// TwinCAT 3 PLC project Main
// ProgramVersion: 3.1.4024.0
// libraries:
//   mobject-core, * (mobject)
//   mobject-graph, * (mobject)
//   mobject-graph-math-pack, * (mobject)
//   mobject-graph-plc-pack, * (mobject)
//   mobject-graph-vision-pack, * (mobject)
//   mobject-server, * (mobject)
//   Tc2_Standard, * (Beckhoff Automation GmbH)
//   Tc2_System, * (Beckhoff Automation GmbH)
//   Tc2_Utilities, * (Beckhoff Automation GmbH)
//   Tc3_Module, * (Beckhoff Automation GmbH)
//   Tc3_Vision, * (Beckhoff Automation GmbH)
// project tree:
//   / PlcTask.TcTTO
//   POUs/Examples/ MyCustomNode.TcPOU, DisplayableImageNode.TcPOU
//   POUs/ MAIN.TcPOU
// real-time tasks:
//   TASK PlcTask: cycle T#10ms, priority 20, ADS port 350

CONFIGURATION Main
    RESOURCE PLC ON TwinCAT3
        TASK PlcTask(INTERVAL := T#10ms, PRIORITY := 20);
        PROGRAM MAIN WITH PlcTask : MAIN;
    END_RESOURCE
END_CONFIGURATION

// ---- POUs/MAIN.TcPOU
PROGRAM MAIN
VAR		

	// installation of the packs is only requried once. 
	initialise: BOOL;
	
	// graph packs
	iecDatatypesPack : IecDatatypesPack; // mobject-graph, 
	plcPack : PlcPack; // mobject-graph-plc-pack
	visionPack : VisionPack; // mobject-graph-vision-pack
	mathPack : MathPack; // mobject-graph-math-pack, this is all packs.  You can also select sub-packs if needed
	
	// custom node
	myCustomNode : MyCustomNode;
	
	// twincat hmi linked variables and nodes
	displayImage1 : ITcVnDisplayableImage;
	displayImage1Node : DisplayableImageNode(displayImage1);
	displayImage2 : ITcVnDisplayableImage;
	displayImage2Node : DisplayableImageNode(displayImage2);
	displayImage3 : ITcVnDisplayableImage;
	displayImage3Node : DisplayableImageNode(displayImage3);

	// application
	graphFramework : GraphFramework;
	server : RpcServer;
	graphFrameworkApi : GraphFrameworkApi(graphFramework);	

END_VAR

IF NOT initialise THEN

	// add graph packs here...
	graphFramework.Install(iecDatatypesPack); // adds primitives such as BOOL, WORD, STRING...
	graphFramework.Install(plcPack); // adds datatypes and nodes base on TC2_Utilities...
	graphFramework.Install(visionPack); // adds datatypes and nodes for TC3_Vision...
	graphFramework.Install(mathPack); // adds all of the math packs.  
	
	// add any custom datatypes here...
	// graphFramework.Datatypes.RegisterDatatype(_customDatatype);
	
	// add any custom nodes here...
	graphFramework.NodeFactory.AddNodeAsPrototype('Custom/MyCustomNode', myCustomNode);

	// add hardware nodes in the same way...
	graphFramework.NodeFactory.AddNodeAsPrototype('Displayable Images/Display Image 1', displayImage1Node);
	graphFramework.NodeFactory.AddNodeAsPrototype('Displayable Images/Display Image 2', displayImage2Node);
	graphFramework.NodeFactory.AddNodeAsPrototype('Displayable Images/Display Image 3', displayImage3Node);
	
	// add the graph framework api to the server, this will register all of the endpoint handlers
	server.RegisterApi(graphFrameworkApi);

	// done
	initialise := TRUE;	

END_IF

// a special feature of .RegisterApi is that the server will know to cyclic call all registered apis each cycle. 
server.CyclicCall();

END_PROGRAM

// ---- POUs/Examples/MyCustomNode.TcPOU
{attribute 'linkalways'} 
{attribute 'no_explicit_call' := 'This FB is a CLASS and must be accessed using methods or properties'}
{attribute 'enable_dynamic_creation'}
FUNCTION_BLOCK MyCustomNode EXTENDS Node
VAR
	myIntParameter : _INT(123);
	myWordParameter : _WORD(456);
	myIntOutput : _INT(0);
	myWordOutput : _WORD(0);
END_VAR

METHOD PUBLIC  Clone : I_Node
VAR_INPUT
END_VAR
VAR
	pNode : POINTER TO MyCustomNode;
END_VAR
pNode := __NEW(MyCustomNode);
Clone := pNode^;
END_METHOD

METHOD FB_init : BOOL
VAR_INPUT
	bInitRetains : BOOL; // if TRUE, the retain variables are initialized (warm start / cold start)
	bInCopyCode : BOOL;  // if TRUE, the instance afterwards gets moved into the copy code (online change)
END_VAR
AddParameter('myIntParam', myIntParameter);
AddParameter('myWordParam', myWordParameter);
AddOutput('myIntOutput', myIntOutput);
AddOutput('myWordOutput', myWordOutput);
END_METHOD

METHOD PROTECTED  OnExecute : HRESULT
myIntOutput.Value := myIntParameter.Value;
myWordOutput.Value := myWordParameter.Value;
END_METHOD

END_FUNCTION_BLOCK

// ---- POUs/Examples/DisplayableImageNode.TcPOU
{attribute 'linkalways'} 
{attribute 'no_explicit_call' := 'This FB is a CLASS and must be accessed using methods or properties'}
{attribute 'enable_dynamic_creation'}
// this node shows you how it is possible to make "hardware nodes", i.e. nodes which are connected to variables which are static.  this
// can be variables linked with the hmi, or could even be i/o pdo
FUNCTION_BLOCK DisplayableImageNode EXTENDS Node
VAR
	ipSrcImage : _ITcVnImage;
	hrPrev : _HRESULT(S_OK);
	ipDestImage : REFERENCE TO ITcVnDisplayableImage;
END_VAR

METHOD PUBLIC  Clone : I_Node
VAR_INPUT
END_VAR
// this node is classed as a hardware node, i.e. there is only one as it is linked to a variable, or I/O point. 
// therefore, when someone tries to clone it, instead of getting a new one, they get the same one. 
Clone := THIS^;
END_METHOD

METHOD PUBLIC Dispose
VAR_INPUT
END_VAR
// you will also add a blank dispose method to prevent the system from automatically destroying the node.  
// hardware nodes are here to stay as they are linked with things in the PLC.
END_METHOD

METHOD FB_init : BOOL
VAR_INPUT
	bInitRetains : BOOL; // if TRUE, the retain variables are initialized (warm start / cold start)
	bInCopyCode : BOOL;  // if TRUE, the instance afterwards gets moved into the copy code (online change)
	DisplayableImage : REFERENCE TO ITcVnDisplayableImage;
END_VAR
ipDestImage REF= DisplayableImage;
AddInput('in', ipSrcImage);
END_METHOD

METHOD PROTECTED  OnExecute : HRESULT
VAR
	result : HRESULT;
END_VAR
result := F_VN_CopyIntoDisplayableImage(ipSrcImage.Value, ipDestImage, hrPrev.Value);

IF succeeded(result) THEN
	// if everything was a success, then leave, the job is done.
	RETURN;
END_IF

// we know that the function failed so we may need to do some tidying

IF ipDestImage = 0 THEN
	// we didn't have a displayable image already, so that's fine.  Nothing to tidy.  Time to leave. 
	RETURN;
END_IF

// we know we have an image, so best is to release it and set the destination to 0. 

ipDestImage.TcRelease();
ipDestImage := 0;
END_METHOD

END_FUNCTION_BLOCK
